// Mitsubishi GX Works2 project: 타이머D저장   PLC: Q02/Q02H

PROGRAM MAIN
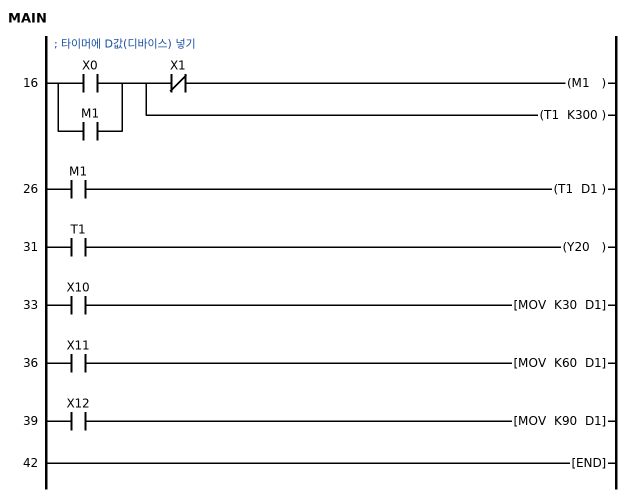
; 타이머에 D값(디바이스) 넣기
16    LD      X0
      OR      M1
      MPS
      ANI     X1
      OUT     M1
      MPP
      OUT     T1 K300
26    LD      M1
      OUT     T1 D1
31    LD      T1
      OUT     Y20
33    LD      X10
      MOV     K30 D1
36    LD      X11
      MOV     K60 D1
39    LD      X12
      MOV     K90 D1
42    END
END_PROGRAM
